INTERFACE I_FileSystemEntry EXTENDS __SYSTEM.IQueryInterface

PROPERTY PUBLIC IsDirectory : BOOL
GET
END_GET
END_PROPERTY

PROPERTY PUBLIC IsFile : BOOL
GET
END_GET
END_PROPERTY

PROPERTY PUBLIC IsNull : BOOL
GET
END_GET
END_PROPERTY

PROPERTY Path : FilePath
GET
END_GET
END_PROPERTY

END_INTERFACE

(* stored: Version 1.1.0.1, ProductVersion 3.1.4024.9
   Itf I_FileSystemEntry: Id {66833fc6-b602-49c7-acc3-7bfa91f32bf6}
   Property IsDirectory: Id {22c81b53-bc65-4de3-b099-f048eca9fcc7}
   Get Get: Id {8ce22853-8680-4574-a632-67e46c1ed9a5}
   Property IsFile: Id {bf38604d-52f0-458b-a7f2-d8a5608712aa}
   Get Get: Id {eab15ada-a806-4d60-b471-b358888d1f84}
   Property IsNull: Id {c7eee129-cfee-4483-ae7c-c99f573df8f7}
   Get Get: Id {27584e77-09aa-4822-9bee-d1c2a73e8907}
   Property Path: Id {e3b1661e-05ad-42dc-91f1-d2ef8175dc30}
   Get Get: Id {a24a2121-dcb9-4ef0-94ed-6232fa627818} *)
